// Mitsubishi GX Works2 project: Genova 14-11-2022_fr   PLC: FX1N/FX1NC

PROGRAM MAIN
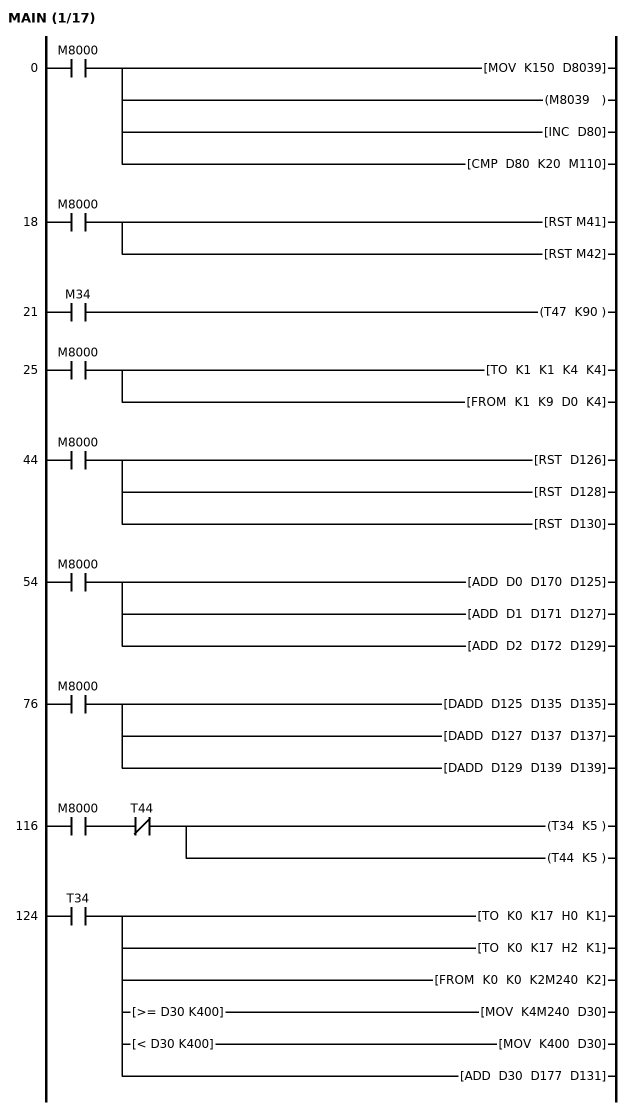
0     LD      M8000
      MOV     K150 D8039
      OUT     M8039
      INC     D80
      CMP     D80 K20 M110
18    LD      M8000
      RST     M41
      RST     M42
21    LD      M34
      OUT     T47 K90
25    LD      M8000
      TO      K1 K1 K4 K4
      FROM    K1 K9 D0 K4
44    LD      M8000
      RST     D126
      RST     D128
      RST     D130
54    LD      M8000
      ADD     D0 D170 D125
      ADD     D1 D171 D127
      ADD     D2 D172 D129
76    LD      M8000
      DADD    D125 D135 D135
      DADD    D127 D137 D137
      DADD    D129 D139 D139
116   LD      M8000
      ANI     T44
      OUT     T34 K5
      OUT     T44 K5
124   LD      T34
      TO      K0 K17 H0 K1
      TO      K0 K17 H2 K1
      FROM    K0 K0 K2M240 K2
      MPS
      AND>=   D30 K400
      MOV     K4M240 D30
      MRD
      AND<    D30 K400
      MOV     K400 D30
      MPP
      ADD     D30 D177 D131
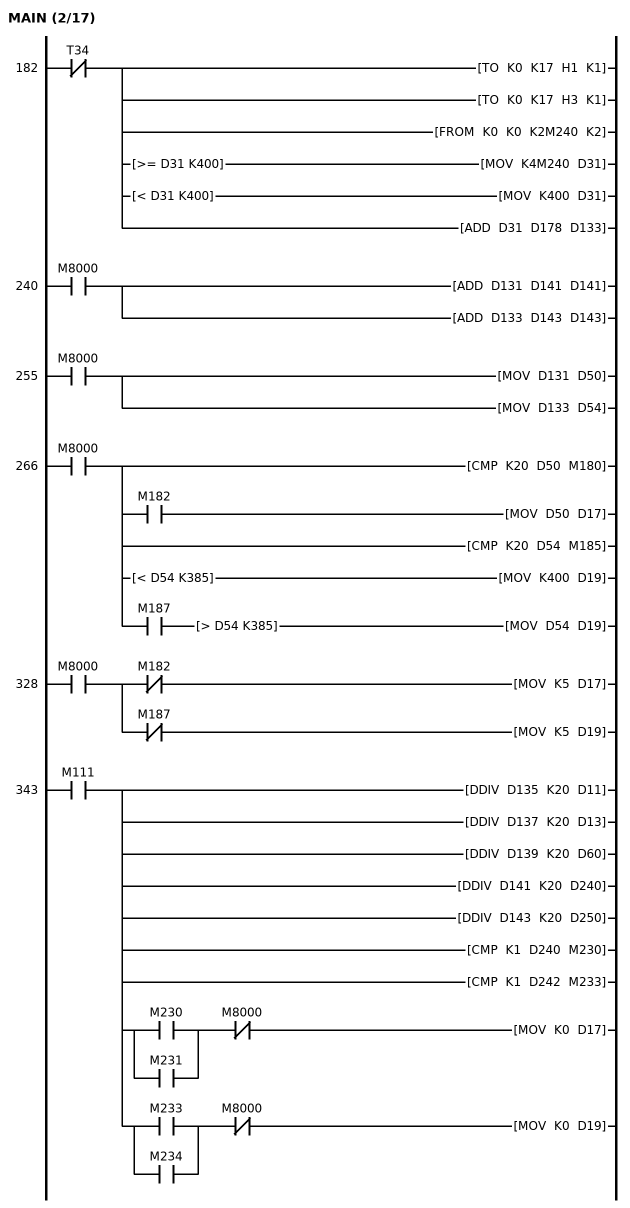
182   LDI     T34
      TO      K0 K17 H1 K1
      TO      K0 K17 H3 K1
      FROM    K0 K0 K2M240 K2
      MPS
      AND>=   D31 K400
      MOV     K4M240 D31
      MRD
      AND<    D31 K400
      MOV     K400 D31
      MPP
      ADD     D31 D178 D133
240   LD      M8000
      ADD     D131 D141 D141
      ADD     D133 D143 D143
255   LD      M8000
      MOV     D131 D50
      MOV     D133 D54
266   LD      M8000
      CMP     K20 D50 M180
      MPS
      AND     M182
      MOV     D50 D17
      MPP
      CMP     K20 D54 M185
      MPS
      AND<    D54 K385
      MOV     K400 D19
      MPP
      AND     M187
      AND>    D54 K385
      MOV     D54 D19
328   LD      M8000
      MPS
      ANI     M182
      MOV     K5 D17
      MPP
      ANI     M187
      MOV     K5 D19
343   LD      M111
      DDIV    D135 K20 D11
      DDIV    D137 K20 D13
      DDIV    D139 K20 D60
      DDIV    D141 K20 D240
      DDIV    D143 K20 D250
      CMP     K1 D240 M230
      CMP     K1 D242 M233
      MPS
      LD      M230
      OR      M231
      ANB
      ANI     M8000
      MOV     K0 D17
      MPP
      LD      M233
      OR      M234
      ANB
      ANI     M8000
      MOV     K0 D19
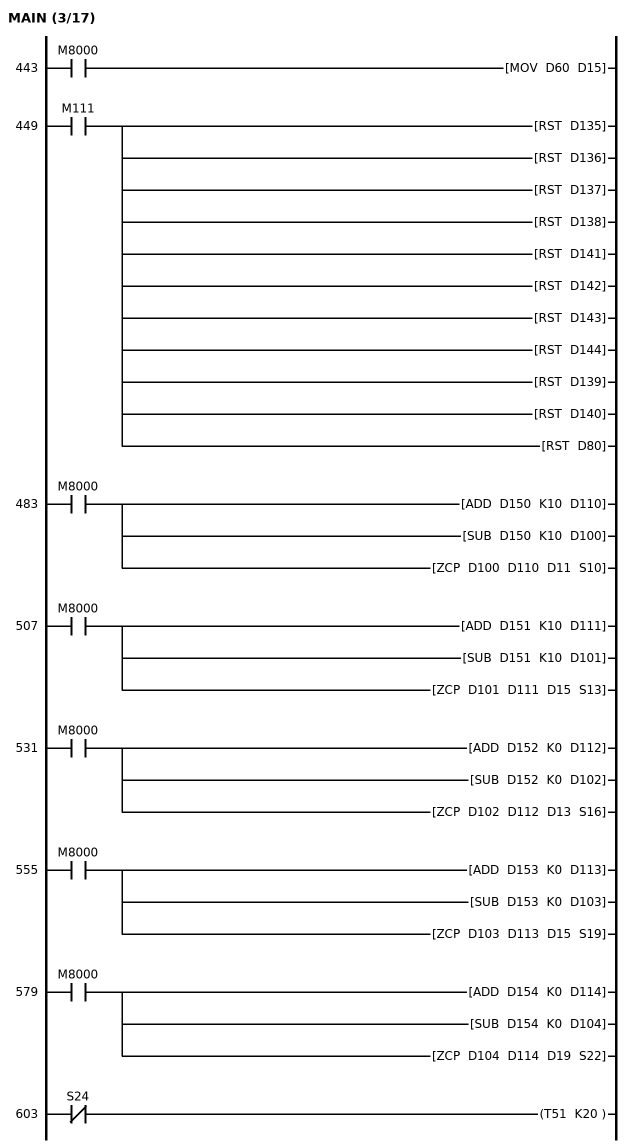
443   LD      M8000
      MOV     D60 D15
449   LD      M111
      RST     D135
      RST     D136
      RST     D137
      RST     D138
      RST     D141
      RST     D142
      RST     D143
      RST     D144
      RST     D139
      RST     D140
      RST     D80
483   LD      M8000
      ADD     D150 K10 D110
      SUB     D150 K10 D100
      ZCP     D100 D110 D11 S10
507   LD      M8000
      ADD     D151 K10 D111
      SUB     D151 K10 D101
      ZCP     D101 D111 D15 S13
531   LD      M8000
      ADD     D152 K0 D112
      SUB     D152 K0 D102
      ZCP     D102 D112 D13 S16
555   LD      M8000
      ADD     D153 K0 D113
      SUB     D153 K0 D103
      ZCP     D103 D113 D15 S19
579   LD      M8000
      ADD     D154 K0 D114
      SUB     D154 K0 D104
      ZCP     D104 D114 D19 S22
603   LDI     S24
      OUT     T51 K20
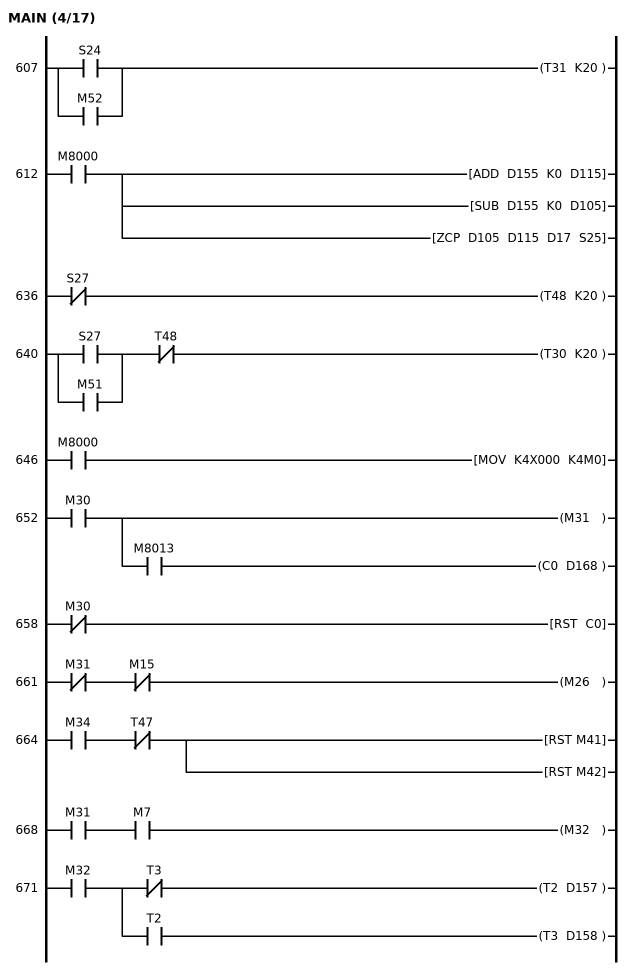
607   LD      S24
      OR      M52
      OUT     T31 K20
612   LD      M8000
      ADD     D155 K0 D115
      SUB     D155 K0 D105
      ZCP     D105 D115 D17 S25
636   LDI     S27
      OUT     T48 K20
640   LD      S27
      OR      M51
      ANI     T48
      OUT     T30 K20
646   LD      M8000
      MOV     K4X000 K4M0
652   LD      M30
      OUT     M31
      AND     M8013
      OUT     C0 D168
658   LDI     M30
      RST     C0
661   LDI     M31
      ANI     M15
      OUT     M26
664   LD      M34
      ANI     T47
      RST     M41
      RST     M42
668   LD      M31
      AND     M7
      OUT     M32
671   LD      M32
      MPS
      ANI     T3
      OUT     T2 D157
      MPP
      AND     T2
      OUT     T3 D158
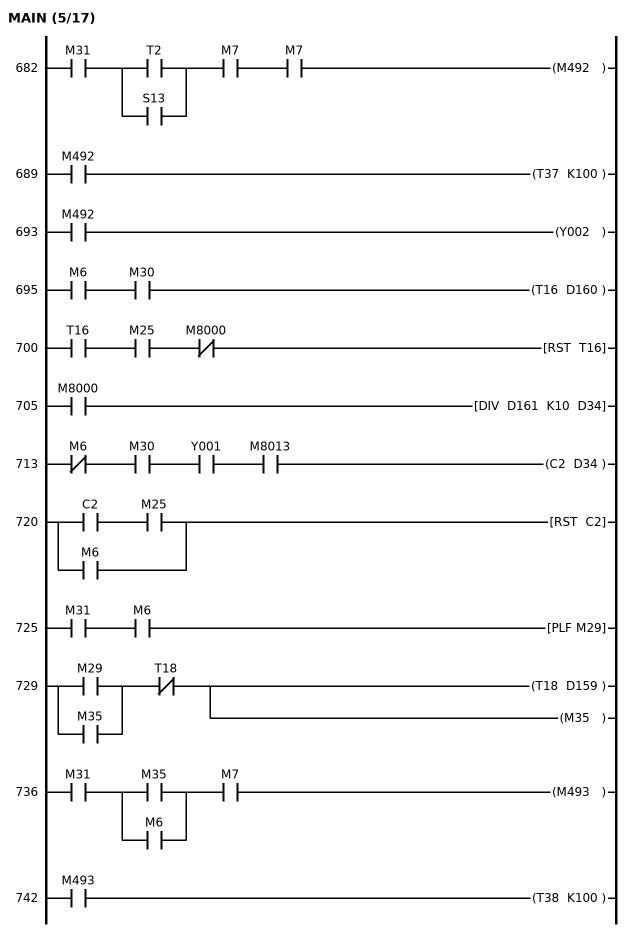
682   LD      M31
      LD      T2
      OR      S13
      ANB
      AND     M7
      AND     M7
      OUT     M492
689   LD      M492
      OUT     T37 K100
693   LD      M492
      OUT     Y002
695   LD      M6
      AND     M30
      OUT     T16 D160
700   LD      T16
      AND     M25
      ANI     M8000
      RST     T16
705   LD      M8000
      DIV     D161 K10 D34
713   LDI     M6
      AND     M30
      AND     Y001
      AND     M8013
      OUT     C2 D34
720   LD      C2
      AND     M25
      OR      M6
      RST     C2
725   LD      M31
      AND     M6
      PLF     M29
729   LD      M29
      OR      M35
      ANI     T18
      OUT     T18 D159
      OUT     M35
736   LD      M31
      LD      M35
      OR      M6
      ANB
      AND     M7
      OUT     M493
742   LD      M493
      OUT     T38 K100
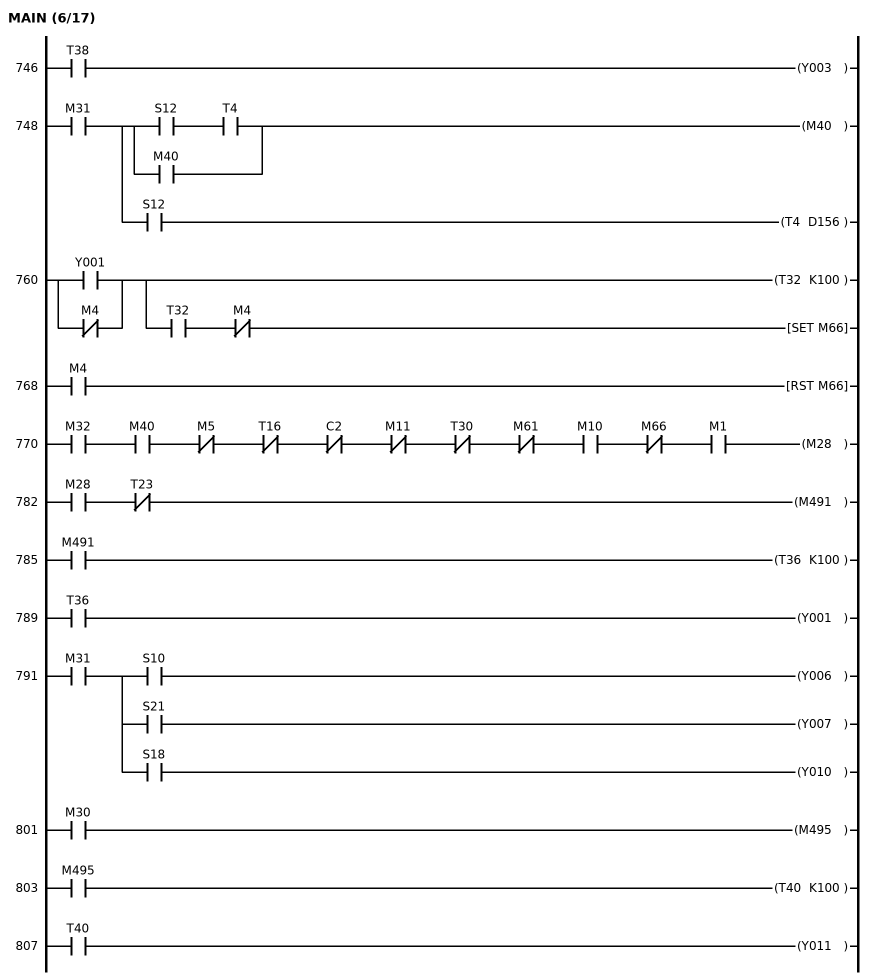
746   LD      T38
      OUT     Y003
748   LD      M31
      MPS
      LD      S12
      AND     T4
      OR      M40
      ANB
      OUT     M40
      MPP
      AND     S12
      OUT     T4 D156
760   LD      Y001
      ORI     M4
      OUT     T32 K100
      AND     T32
      ANI     M4
      SET     M66
768   LD      M4
      RST     M66
770   LD      M32
      AND     M40
      ANI     M5
      ANI     T16
      ANI     C2
      ANI     M11
      ANI     T30
      ANI     M61
      AND     M10
      ANI     M66
      AND     M1
      OUT     M28
782   LD      M28
      ANI     T23
      OUT     M491
785   LD      M491
      OUT     T36 K100
789   LD      T36
      OUT     Y001
791   LD      M31
      MPS
      AND     S10
      OUT     Y006
      MRD
      AND     S21
      OUT     Y007
      MPP
      AND     S18
      OUT     Y010
801   LD      M30
      OUT     M495
803   LD      M495
      OUT     T40 K100
807   LD      T40
      OUT     Y011
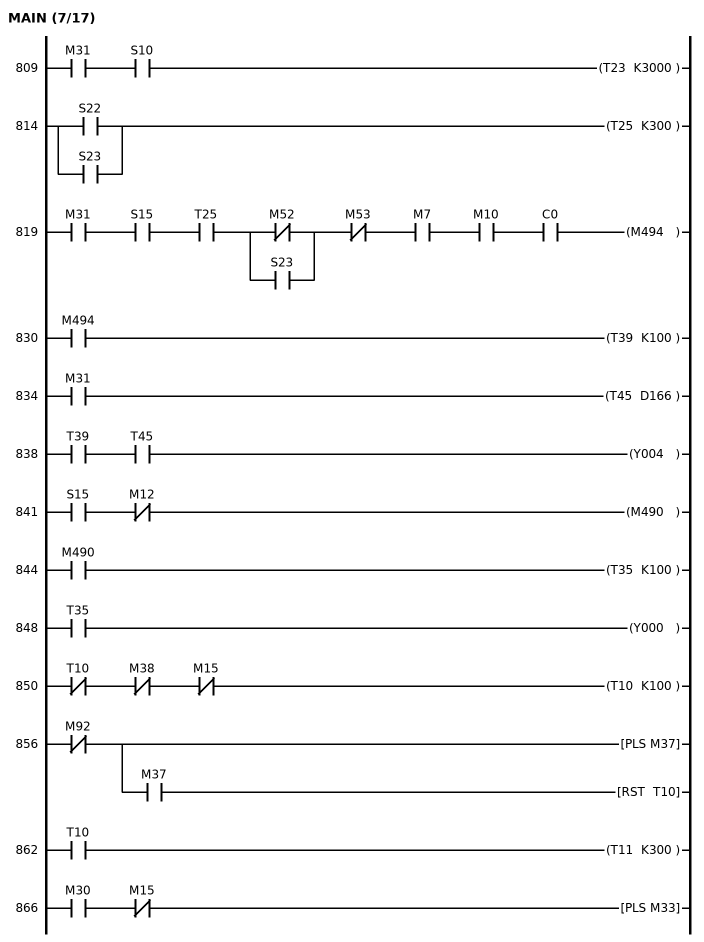
809   LD      M31
      AND     S10
      OUT     T23 K3000
814   LD      S22
      OR      S23
      OUT     T25 K300
819   LD      M31
      AND     S15
      AND     T25
      LDI     M52
      OR      S23
      ANB
      ANI     M53
      AND     M7
      AND     M10
      AND     C0
      OUT     M494
830   LD      M494
      OUT     T39 K100
834   LD      M31
      OUT     T45 D166
838   LD      T39
      AND     T45
      OUT     Y004
841   LD      S15
      ANI     M12
      OUT     M490
844   LD      M490
      OUT     T35 K100
848   LD      T35
      OUT     Y000
850   LDI     T10
      ANI     M38
      ANI     M15
      OUT     T10 K100
856   LDI     M92
      PLS     M37
      AND     M37
      RST     T10
862   LD      T10
      OUT     T11 K300
866   LD      M30
      ANI     M15
      PLS     M33
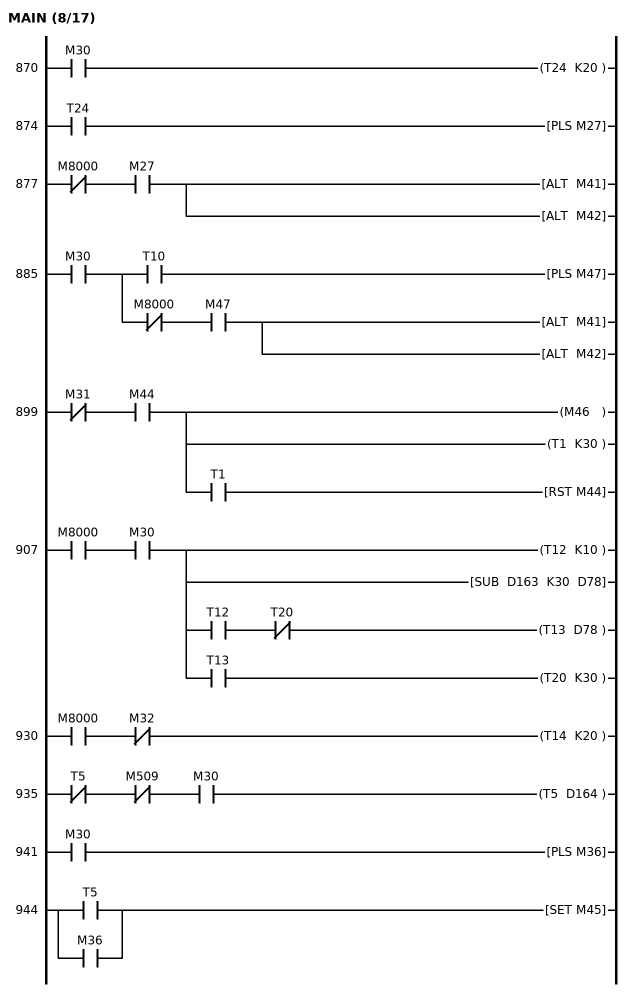
870   LD      M30
      OUT     T24 K20
874   LD      T24
      PLS     M27
877   LDI     M8000
      AND     M27
      ALT     M41
      ALT     M42
885   LD      M30
      MPS
      AND     T10
      PLS     M47
      MPP
      ANI     M8000
      AND     M47
      ALT     M41
      ALT     M42
899   LDI     M31
      AND     M44
      OUT     M46
      OUT     T1 K30
      AND     T1
      RST     M44
907   LD      M8000
      AND     M30
      OUT     T12 K10
      SUB     D163 K30 D78
      MPS
      AND     T12
      ANI     T20
      OUT     T13 D78
      MPP
      AND     T13
      OUT     T20 K30
930   LD      M8000
      ANI     M32
      OUT     T14 K20
935   LDI     T5
      ANI     M509
      AND     M30
      OUT     T5 D164
941   LD      M30
      PLS     M36
944   LD      T5
      OR      M36
      SET     M45
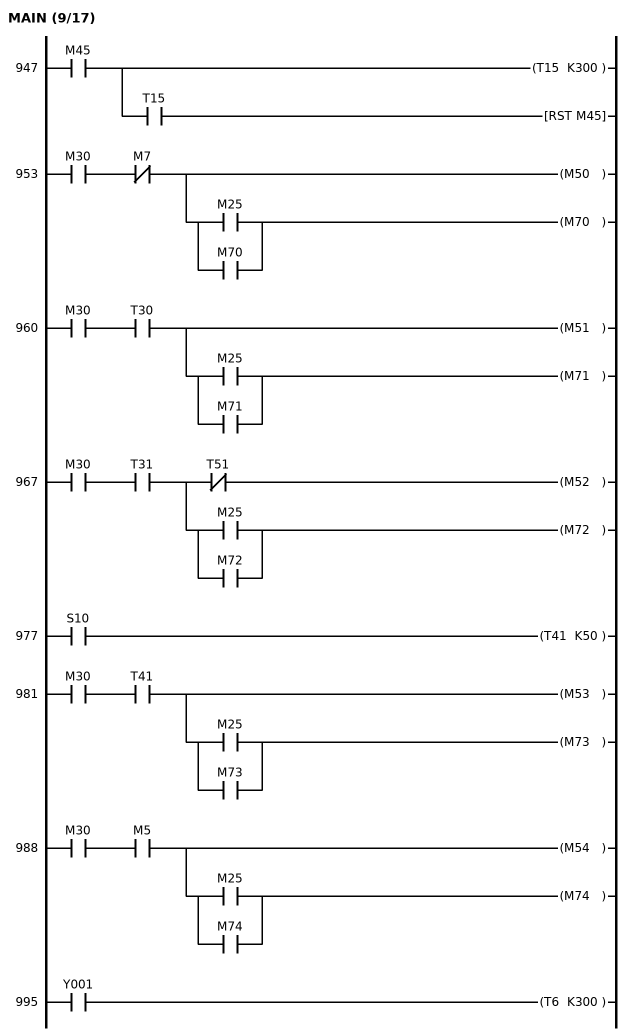
947   LD      M45
      OUT     T15 K300
      AND     T15
      RST     M45
953   LD      M30
      ANI     M7
      OUT     M50
      LD      M25
      OR      M70
      ANB
      OUT     M70
960   LD      M30
      AND     T30
      OUT     M51
      LD      M25
      OR      M71
      ANB
      OUT     M71
967   LD      M30
      AND     T31
      MPS
      ANI     T51
      OUT     M52
      MPP
      LD      M25
      OR      M72
      ANB
      OUT     M72
977   LD      S10
      OUT     T41 K50
981   LD      M30
      AND     T41
      OUT     M53
      LD      M25
      OR      M73
      ANB
      OUT     M73
988   LD      M30
      AND     M5
      OUT     M54
      LD      M25
      OR      M74
      ANB
      OUT     M74
995   LD      Y001
      OUT     T6 K300
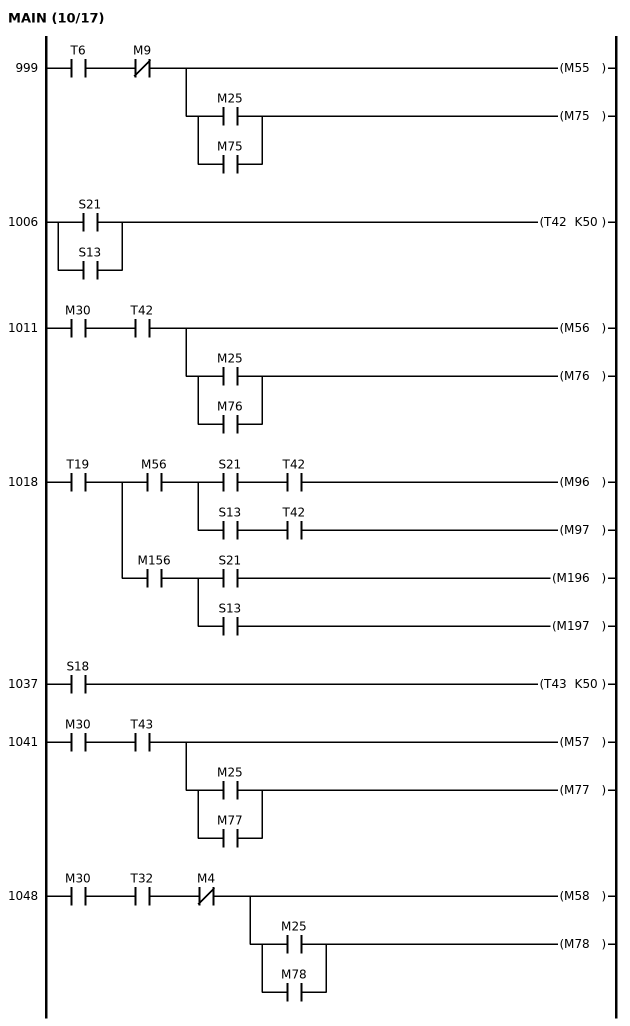
999   LD      T6
      ANI     M9
      OUT     M55
      LD      M25
      OR      M75
      ANB
      OUT     M75
1006  LD      S21
      OR      S13
      OUT     T42 K50
1011  LD      M30
      AND     T42
      OUT     M56
      LD      M25
      OR      M76
      ANB
      OUT     M76
1018  LD      T19
      MPS
      AND     M56
      MPS
      AND     S21
      AND     T42
      OUT     M96
      MPP
      AND     S13
      AND     T42
      OUT     M97
      MPP
      AND     M156
      MPS
      AND     S21
      OUT     M196
      MPP
      AND     S13
      OUT     M197
1037  LD      S18
      OUT     T43 K50
1041  LD      M30
      AND     T43
      OUT     M57
      LD      M25
      OR      M77
      ANB
      OUT     M77
1048  LD      M30
      AND     T32
      ANI     M4
      OUT     M58
      LD      M25
      OR      M78
      ANB
      OUT     M78
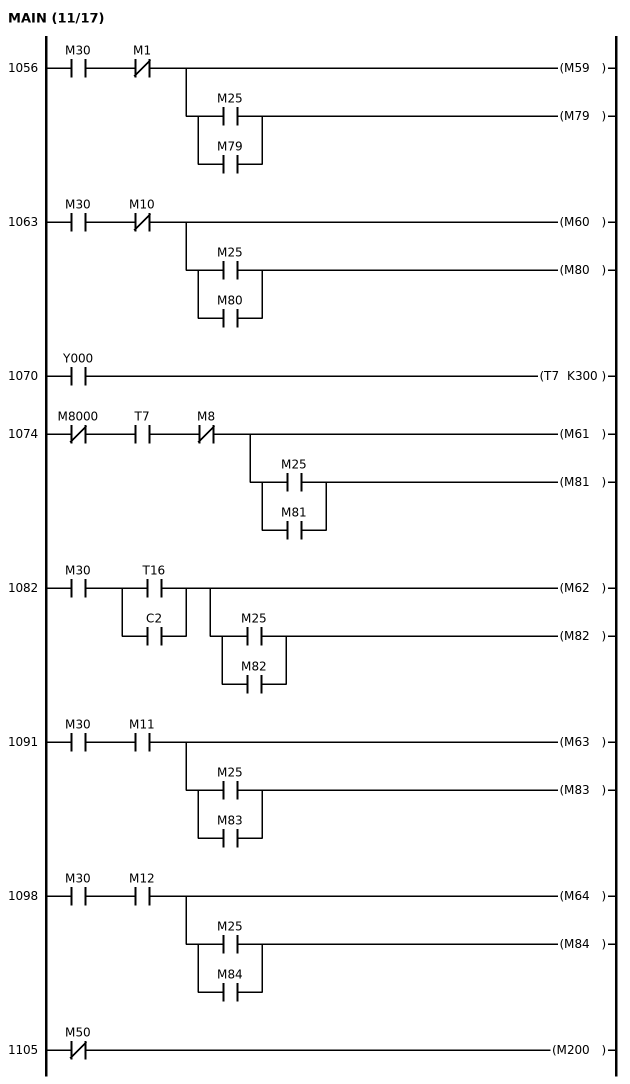
1056  LD      M30
      ANI     M1
      OUT     M59
      LD      M25
      OR      M79
      ANB
      OUT     M79
1063  LD      M30
      ANI     M10
      OUT     M60
      LD      M25
      OR      M80
      ANB
      OUT     M80
1070  LD      Y000
      OUT     T7 K300
1074  LDI     M8000
      AND     T7
      ANI     M8
      OUT     M61
      LD      M25
      OR      M81
      ANB
      OUT     M81
1082  LD      M30
      LD      T16
      OR      C2
      ANB
      OUT     M62
      LD      M25
      OR      M82
      ANB
      OUT     M82
1091  LD      M30
      AND     M11
      OUT     M63
      LD      M25
      OR      M83
      ANB
      OUT     M83
1098  LD      M30
      AND     M12
      OUT     M64
      LD      M25
      OR      M84
      ANB
      OUT     M84
1105  LDI     M50
      OUT     M200
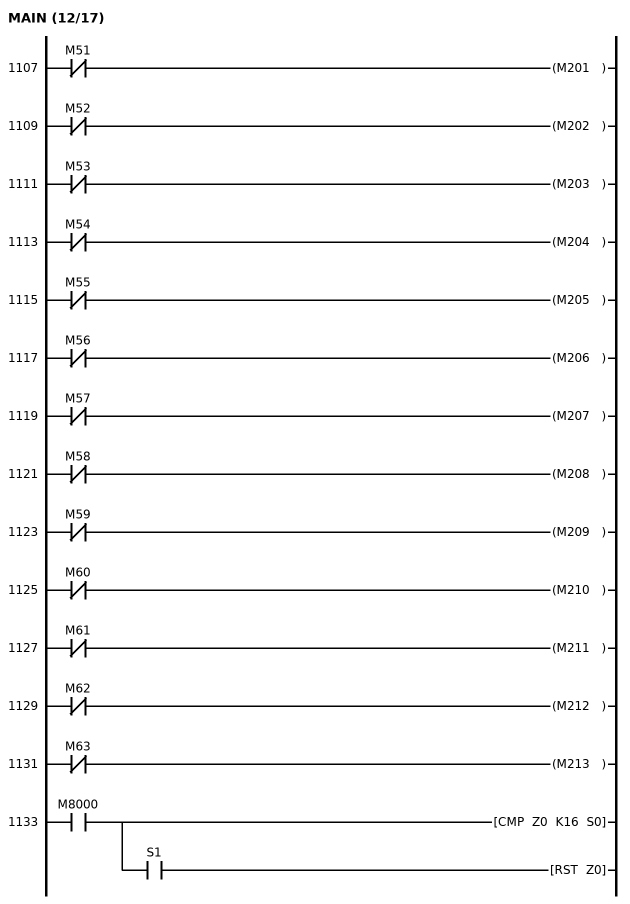
1107  LDI     M51
      OUT     M201
1109  LDI     M52
      OUT     M202
1111  LDI     M53
      OUT     M203
1113  LDI     M54
      OUT     M204
1115  LDI     M55
      OUT     M205
1117  LDI     M56
      OUT     M206
1119  LDI     M57
      OUT     M207
1121  LDI     M58
      OUT     M208
1123  LDI     M59
      OUT     M209
1125  LDI     M60
      OUT     M210
1127  LDI     M61
      OUT     M211
1129  LDI     M62
      OUT     M212
1131  LDI     M63
      OUT     M213
1133  LD      M8000
      CMP     Z0 K16 S0
      AND     S1
      RST     Z0
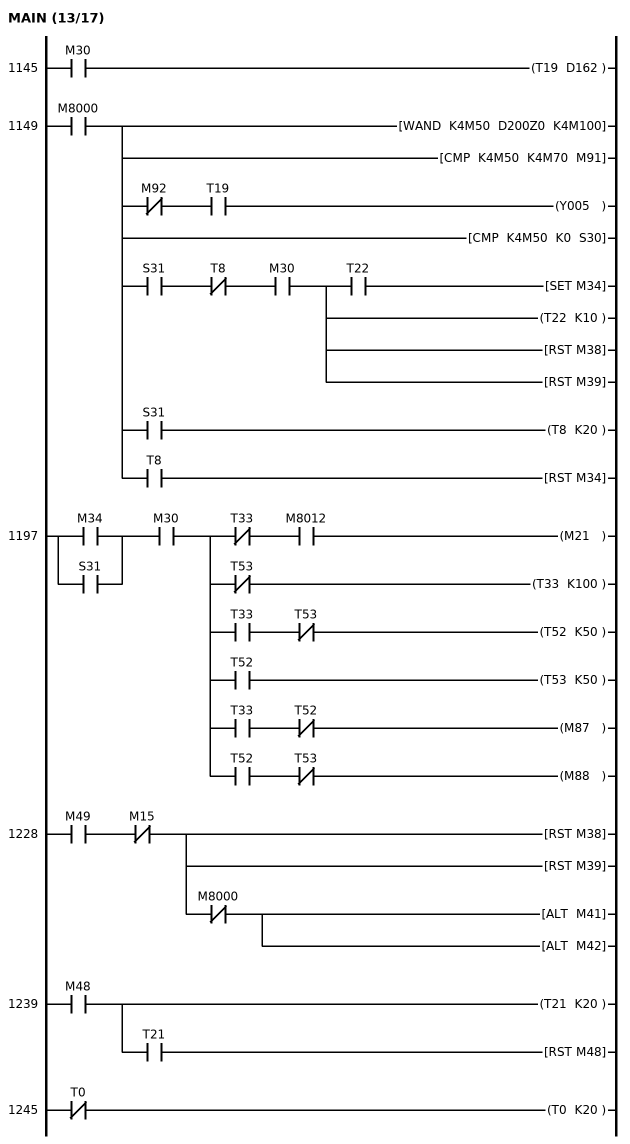
1145  LD      M30
      OUT     T19 D162
1149  LD      M8000
      WAND    K4M50 D200Z0 K4M100
      CMP     K4M50 K4M70 M91
      MPS
      ANI     M92
      AND     T19
      OUT     Y005
      MPP
      CMP     K4M50 K0 S30
      MPS
      AND     S31
      ANI     T8
      AND     M30
      MPS
      AND     T22
      SET     M34
      MPP
      OUT     T22 K10
      RST     M38
      RST     M39
      MRD
      AND     S31
      OUT     T8 K20
      MPP
      AND     T8
      RST     M34
1197  LD      M34
      OR      S31
      AND     M30
      MPS
      ANI     T33
      AND     M8012
      OUT     M21
      MRD
      ANI     T53
      OUT     T33 K100
      MRD
      AND     T33
      ANI     T53
      OUT     T52 K50
      MRD
      AND     T52
      OUT     T53 K50
      MRD
      AND     T33
      ANI     T52
      OUT     M87
      MPP
      AND     T52
      ANI     T53
      OUT     M88
1228  LD      M49
      ANI     M15
      RST     M38
      RST     M39
      ANI     M8000
      ALT     M41
      ALT     M42
1239  LD      M48
      OUT     T21 K20
      AND     T21
      RST     M48
1245  LDI     T0
      OUT     T0 K20
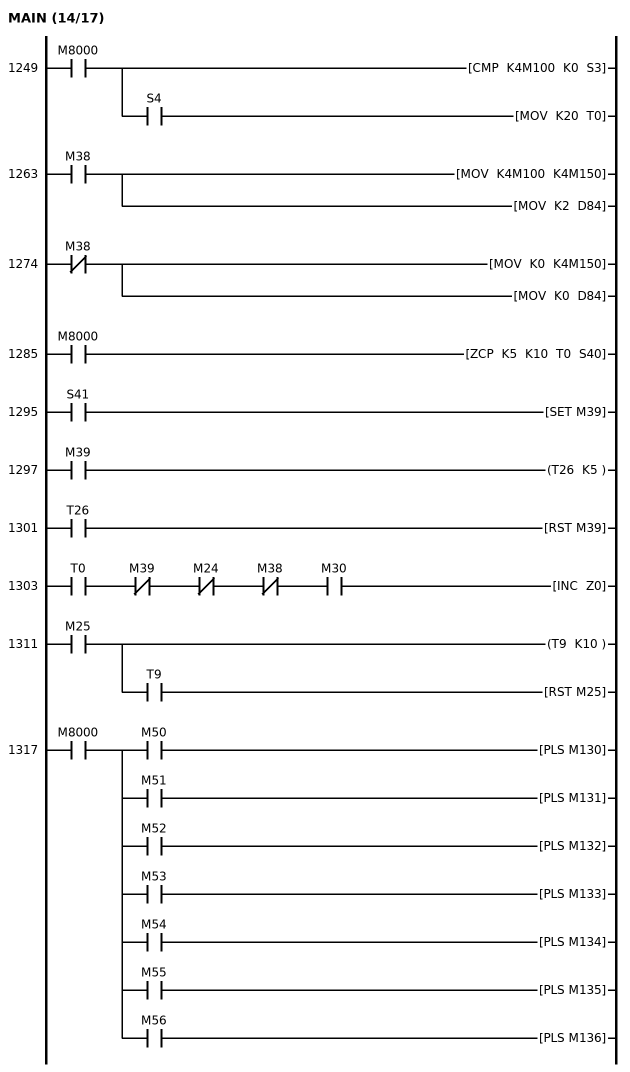
1249  LD      M8000
      CMP     K4M100 K0 S3
      AND     S4
      MOV     K20 T0
1263  LD      M38
      MOV     K4M100 K4M150
      MOV     K2 D84
1274  LDI     M38
      MOV     K0 K4M150
      MOV     K0 D84
1285  LD      M8000
      ZCP     K5 K10 T0 S40
1295  LD      S41
      SET     M39
1297  LD      M39
      OUT     T26 K5
1301  LD      T26
      RST     M39
1303  LD      T0
      ANI     M39
      ANI     M24
      ANI     M38
      AND     M30
      INC     Z0
1311  LD      M25
      OUT     T9 K10
      AND     T9
      RST     M25
1317  LD      M8000
      MPS
      AND     M50
      PLS     M130
      MRD
      AND     M51
      PLS     M131
      MRD
      AND     M52
      PLS     M132
      MRD
      AND     M53
      PLS     M133
      MRD
      AND     M54
      PLS     M134
      MRD
      AND     M55
      PLS     M135
      MPP
      AND     M56
      PLS     M136
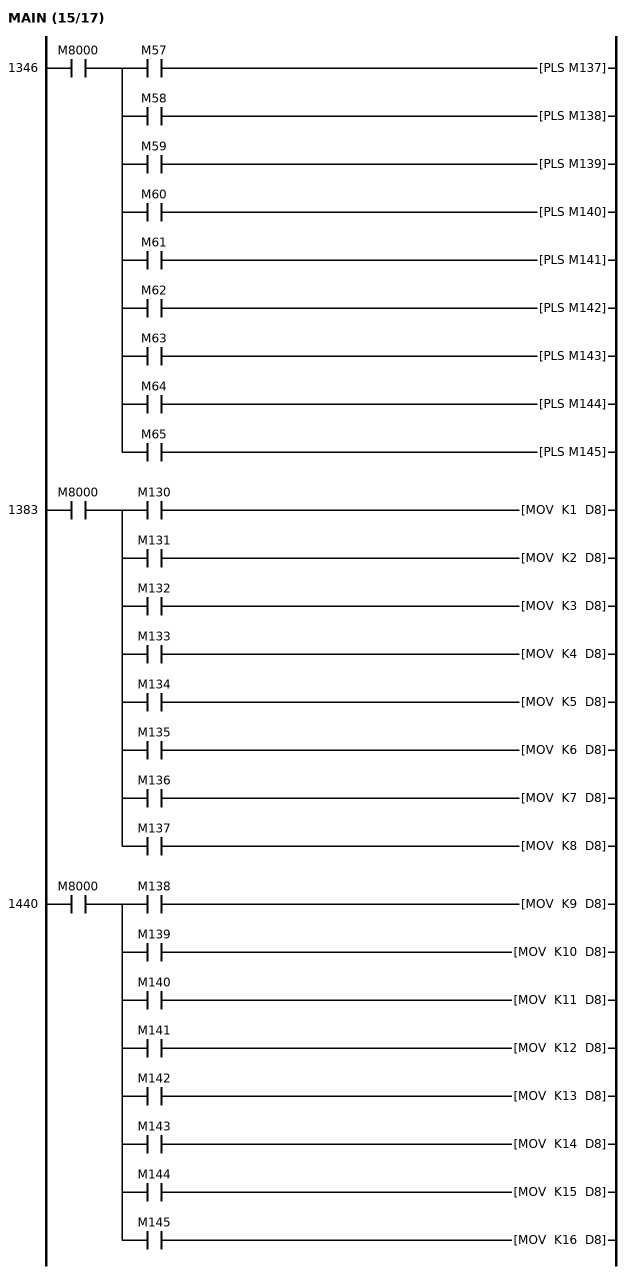
1346  LD      M8000
      MPS
      AND     M57
      PLS     M137
      MRD
      AND     M58
      PLS     M138
      MRD
      AND     M59
      PLS     M139
      MRD
      AND     M60
      PLS     M140
      MRD
      AND     M61
      PLS     M141
      MRD
      AND     M62
      PLS     M142
      MRD
      AND     M63
      PLS     M143
      MRD
      AND     M64
      PLS     M144
      MPP
      AND     M65
      PLS     M145
1383  LD      M8000
      MPS
      AND     M130
      MOV     K1 D8
      MRD
      AND     M131
      MOV     K2 D8
      MRD
      AND     M132
      MOV     K3 D8
      MRD
      AND     M133
      MOV     K4 D8
      MRD
      AND     M134
      MOV     K5 D8
      MRD
      AND     M135
      MOV     K6 D8
      MRD
      AND     M136
      MOV     K7 D8
      MPP
      AND     M137
      MOV     K8 D8
1440  LD      M8000
      MPS
      AND     M138
      MOV     K9 D8
      MRD
      AND     M139
      MOV     K10 D8
      MRD
      AND     M140
      MOV     K11 D8
      MRD
      AND     M141
      MOV     K12 D8
      MRD
      AND     M142
      MOV     K13 D8
      MRD
      AND     M143
      MOV     K14 D8
      MRD
      AND     M144
      MOV     K15 D8
      MPP
      AND     M145
      MOV     K16 D8
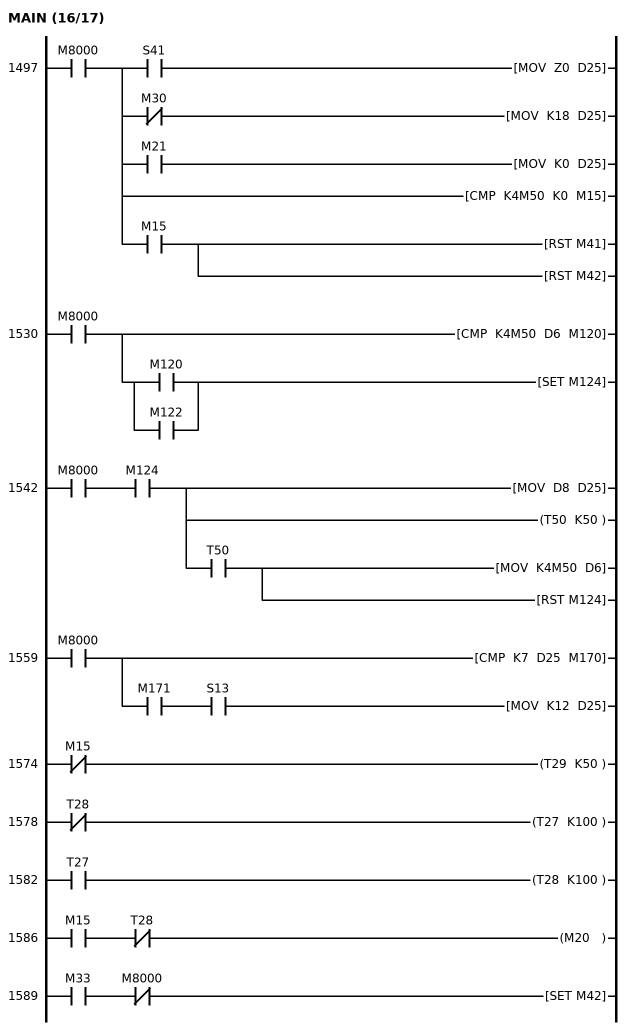
1497  LD      M8000
      MPS
      AND     S41
      MOV     Z0 D25
      MRD
      ANI     M30
      MOV     K18 D25
      MRD
      AND     M21
      MOV     K0 D25
      MPP
      CMP     K4M50 K0 M15
      AND     M15
      RST     M41
      RST     M42
1530  LD      M8000
      CMP     K4M50 D6 M120
      LD      M120
      OR      M122
      ANB
      SET     M124
1542  LD      M8000
      AND     M124
      MOV     D8 D25
      OUT     T50 K50
      AND     T50
      MOV     K4M50 D6
      RST     M124
1559  LD      M8000
      CMP     K7 D25 M170
      AND     M171
      AND     S13
      MOV     K12 D25
1574  LDI     M15
      OUT     T29 K50
1578  LDI     T28
      OUT     T27 K100
1582  LD      T27
      OUT     T28 K100
1586  LD      M15
      ANI     T28
      OUT     M20
1589  LD      M33
      ANI     M8000
      SET     M42
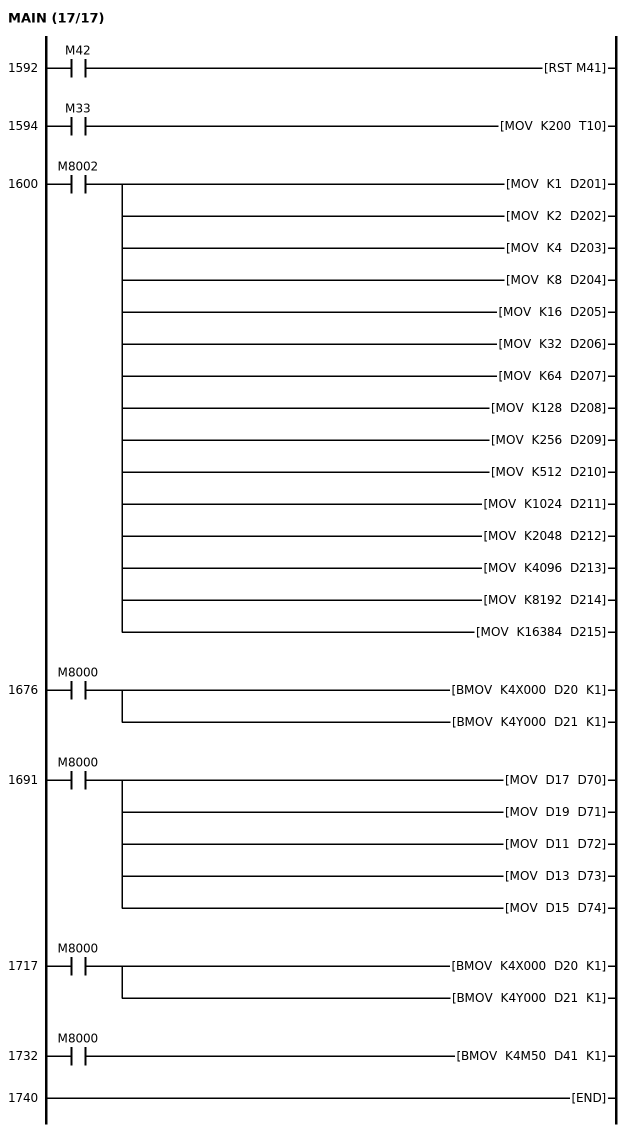
1592  LD      M42
      RST     M41
1594  LD      M33
      MOV     K200 T10
1600  LD      M8002
      MOV     K1 D201
      MOV     K2 D202
      MOV     K4 D203
      MOV     K8 D204
      MOV     K16 D205
      MOV     K32 D206
      MOV     K64 D207
      MOV     K128 D208
      MOV     K256 D209
      MOV     K512 D210
      MOV     K1024 D211
      MOV     K2048 D212
      MOV     K4096 D213
      MOV     K8192 D214
      MOV     K16384 D215
1676  LD      M8000
      BMOV    K4X000 D20 K1
      BMOV    K4Y000 D21 K1
1691  LD      M8000
      MOV     D17 D70
      MOV     D19 D71
      MOV     D11 D72
      MOV     D13 D73
      MOV     D15 D74
1717  LD      M8000
      BMOV    K4X000 D20 K1
      BMOV    K4Y000 D21 K1
1732  LD      M8000
      BMOV    K4M50 D41 K1
1740  END
END_PROGRAM
